// Mitsubishi GX Works2 project: 0926최신화dev   PLC: Q02U

PROGRAM INPUT
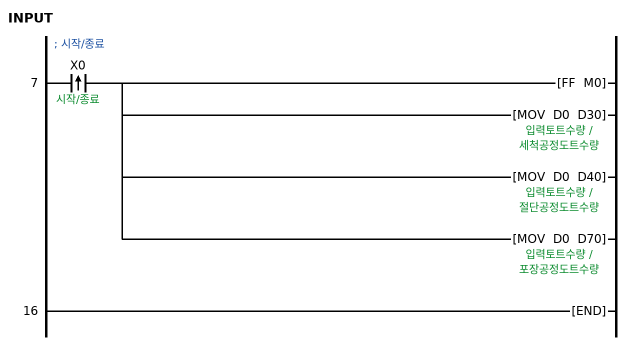
; 시작/종료
7     LDP     X0  ; 시작/종료
      FF      M0
      MOV     D0 D30  ; 입력토트수량 / 세척공정도트수량
      MOV     D0 D40  ; 절단공정도트수량
      MOV     D0 D70  ; 포장공정도트수량
16    END
END_PROGRAM

PROGRAM 세척공정
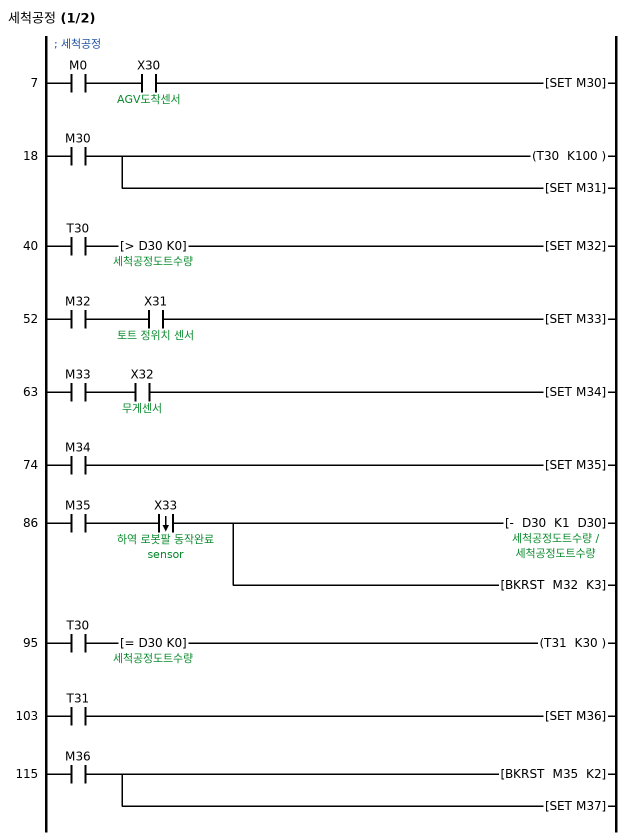
; 세척공정
7     LD      M0
      AND     X30  ; AGV도착센서
      SET     M30
        [note] 펌프모터 ON
18    LD      M30
      OUT     T30 K100
        [note] 펌핑모터 OFF
      SET     M31
        [note] SubCVY ON
40    LD      T30
      AND>    D30 K0  ; 세척공정도트수량
      SET     M32
        [note] 토트 발생
52    LD      M32
      AND     X31  ; 토트 정위치 센서
      SET     M33
        [note] MainCVY ON
63    LD      M33
      AND     X32  ; 무게센서
      SET     M34
        [note] MainCVY OFF
74    LD      M34
      SET     M35
        [note] 하역 로봇팔 ON
86    LD      M35
      ANDF    X33  ; 하역 로봇팔 동작완료 sensor
      -       D30 K1 D30
      BKRST   M32 K3
95    LD      T30
      AND=    D30 K0  ; 세척공정도트수량
      OUT     T31 K30
103   LD      T31
      SET     M36
        [note] 하역 로봇팔 OFF
115   LD      M36
      BKRST   M35 K2
      SET     M37
        [note] AGV 다음 공정 이동, SubCVY OFF
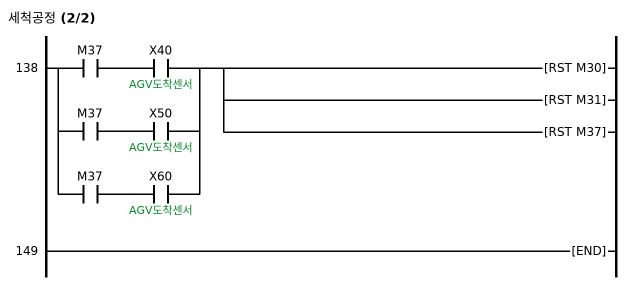
138   LD      M37
      AND     X40  ; AGV도착센서
      LD      M37
      AND     X50  ; AGV도착센서
      ORB
      LD      M37
      AND     X60  ; AGV도착센서
      ORB
      RST     M30
      RST     M31
      RST     M37
149   END
END_PROGRAM

PROGRAM 열풍건조
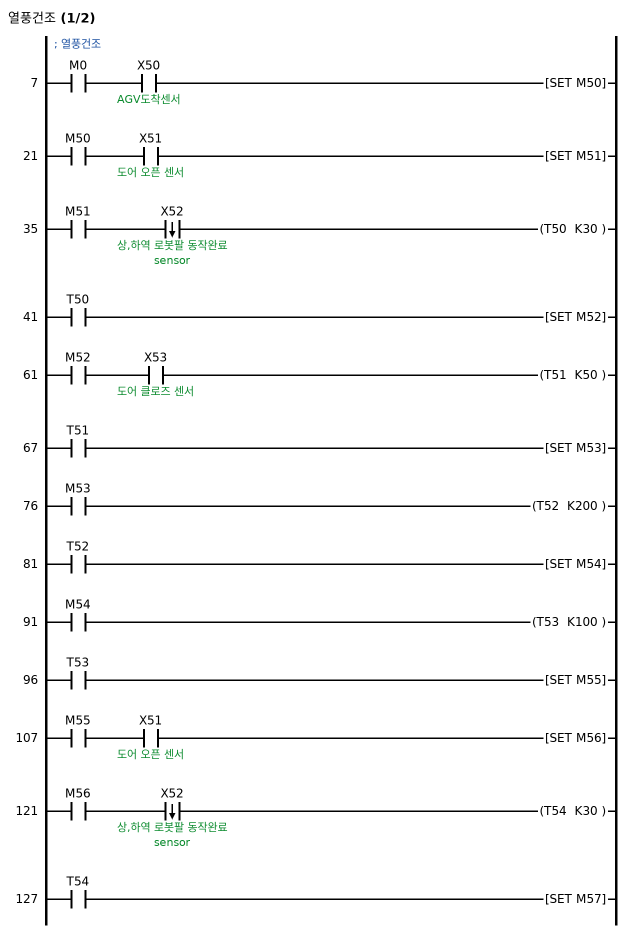
; 열풍건조
7     LD      M0
      AND     X50  ; AGV도착센서
      SET     M50
        [note] 도어 오픈모터(정)
21    LD      M50
      AND     X51  ; 도어 오픈 센서
      SET     M51
        [note] 상역 로봇 팔동작
35    LD      M51
      ANDF    X52  ; 상,하역 로봇팔 동작완료 sensor
      OUT     T50 K30
41    LD      T50
      SET     M52
        [note] 도어 클로즈모터(정), 로봇팔 OFF
61    LD      M52
      AND     X53  ; 도어 클로즈 센서
      OUT     T51 K50
67    LD      T51
      SET     M53
        [note] 건조기 ON
76    LD      M53
      OUT     T52 K200
81    LD      T52
      SET     M54
        [note] 건조기 OFF
91    LD      M54
      OUT     T53 K100
96    LD      T53
      SET     M55
        [note] 도어 오픈CYL
107   LD      M55
      AND     X51  ; 도어 오픈 센서
      SET     M56
        [note] 하역 로봇팔 동작
121   LD      M56
      ANDF    X52  ; 상,하역 로봇팔 동작완료 sensor
      OUT     T54 K30
127   LD      T54
      SET     M57
        [note] 도어 클로즈CYL, 로봇팔 OFF
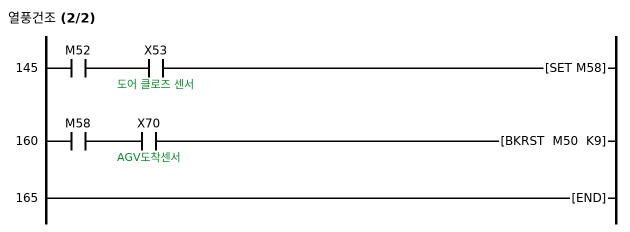
145   LD      M52
      AND     X53  ; 도어 클로즈 센서
      SET     M58
        [note] AGV 다음 공정 이동
160   LD      M58
      AND     X70  ; AGV도착센서
      BKRST   M50 K9
165   END
END_PROGRAM

PROGRAM OUTPUT
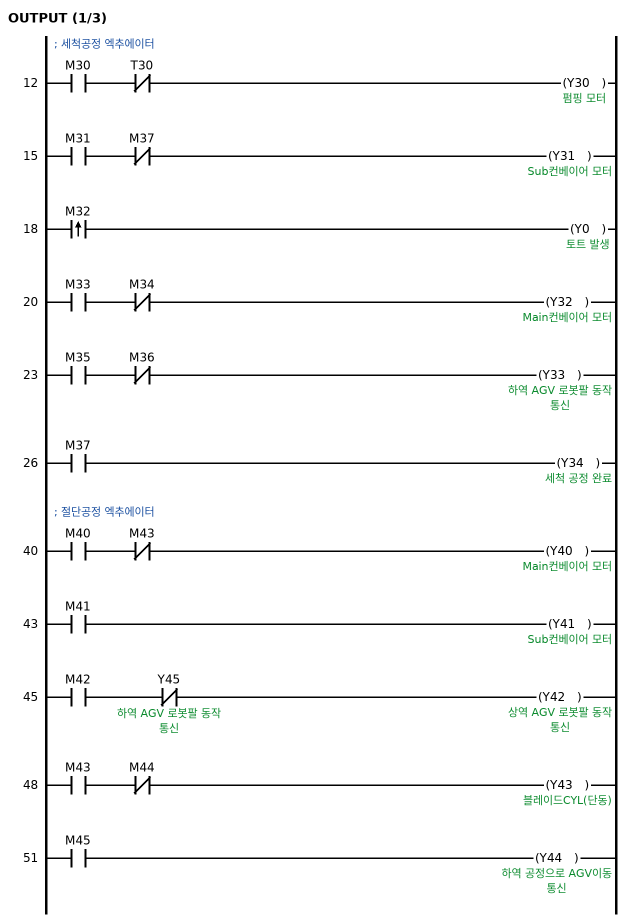
; 세척공정 엑추에이터
12    LD      M30
      ANI     T30
      OUT     Y30  ; 펌핑 모터
15    LD      M31
      ANI     M37
      OUT     Y31  ; Sub컨베이어 모터
18    LDP     M32
      OUT     Y0  ; 토트 발생
20    LD      M33
      ANI     M34
      OUT     Y32  ; Main컨베이어 모터
23    LD      M35
      ANI     M36
      OUT     Y33  ; 하역 AGV 로봇팔 동작 통신
26    LD      M37
      OUT     Y34  ; 세척 공정 완료
; 절단공정 엑추에이터
40    LD      M40
      ANI     M43
      OUT     Y40  ; Main컨베이어 모터
43    LD      M41
      OUT     Y41  ; Sub컨베이어 모터
45    LD      M42
      ANI     Y45  ; 하역 AGV 로봇팔 동작 통신
      OUT     Y42  ; 상역 AGV 로봇팔 동작 통신
48    LD      M43
      ANI     M44
      OUT     Y43  ; 블레이드CYL(단동)
51    LD      M45
      OUT     Y44  ; 하역 공정으로 AGV이동 통신
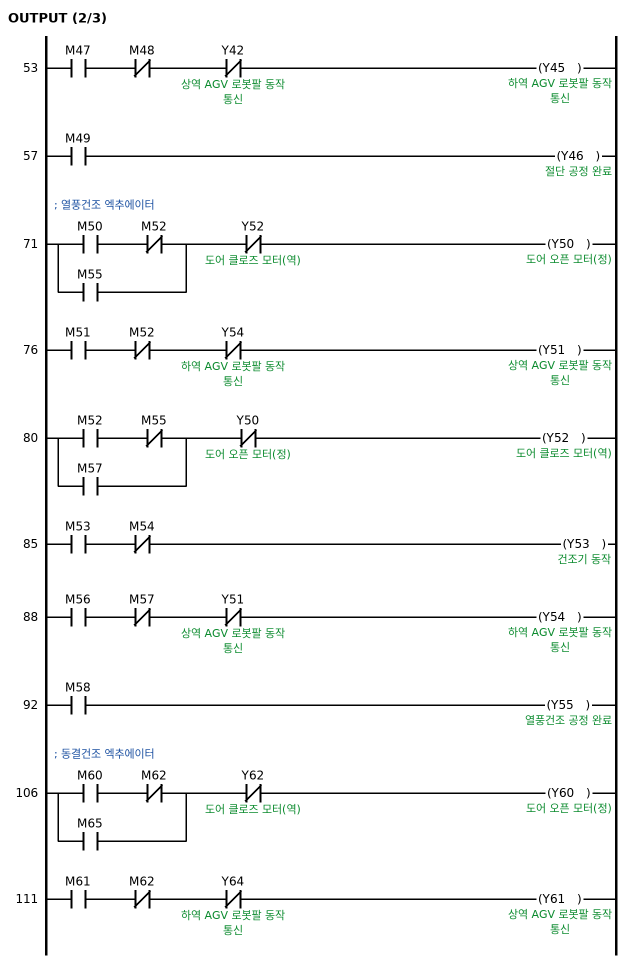
53    LD      M47
      ANI     M48
      ANI     Y42  ; 상역 AGV 로봇팔 동작 통신
      OUT     Y45  ; 하역 AGV 로봇팔 동작 통신
57    LD      M49
      OUT     Y46  ; 절단 공정 완료
; 열풍건조 엑추에이터
71    LD      M50
      ANI     M52
      OR      M55
      ANI     Y52  ; 도어 클로즈 모터(역)
      OUT     Y50  ; 도어 오픈 모터(정)
76    LD      M51
      ANI     M52
      ANI     Y54  ; 하역 AGV 로봇팔 동작 통신
      OUT     Y51  ; 상역 AGV 로봇팔 동작 통신
80    LD      M52
      ANI     M55
      OR      M57
      ANI     Y50  ; 도어 오픈 모터(정)
      OUT     Y52  ; 도어 클로즈 모터(역)
85    LD      M53
      ANI     M54
      OUT     Y53  ; 건조기 동작
88    LD      M56
      ANI     M57
      ANI     Y51  ; 상역 AGV 로봇팔 동작 통신
      OUT     Y54  ; 하역 AGV 로봇팔 동작 통신
92    LD      M58
      OUT     Y55  ; 열풍건조 공정 완료
; 동결건조 엑추에이터
106   LD      M60
      ANI     M62
      OR      M65
      ANI     Y62  ; 도어 클로즈 모터(역)
      OUT     Y60  ; 도어 오픈 모터(정)
111   LD      M61
      ANI     M62
      ANI     Y64  ; 하역 AGV 로봇팔 동작 통신
      OUT     Y61  ; 상역 AGV 로봇팔 동작 통신
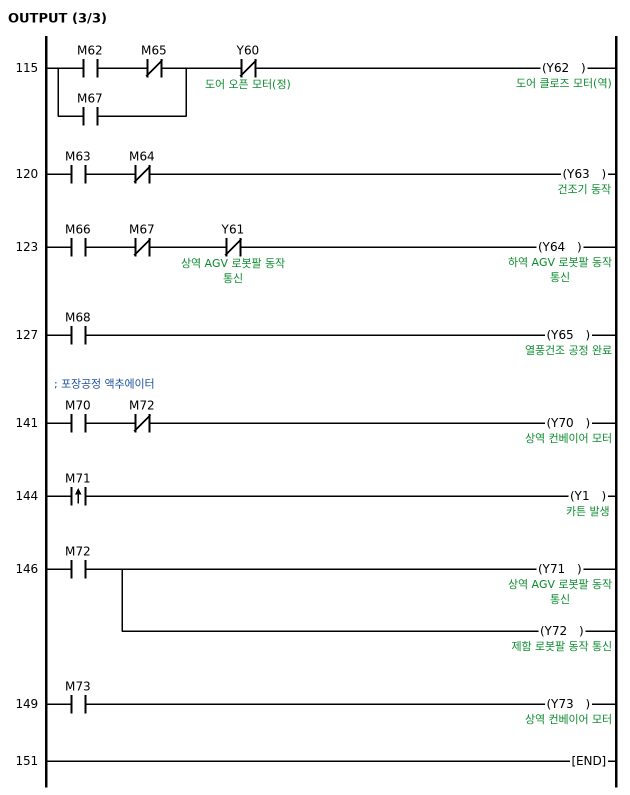
115   LD      M62
      ANI     M65
      OR      M67
      ANI     Y60  ; 도어 오픈 모터(정)
      OUT     Y62  ; 도어 클로즈 모터(역)
120   LD      M63
      ANI     M64
      OUT     Y63  ; 건조기 동작
123   LD      M66
      ANI     M67
      ANI     Y61  ; 상역 AGV 로봇팔 동작 통신
      OUT     Y64  ; 하역 AGV 로봇팔 동작 통신
127   LD      M68
      OUT     Y65  ; 열풍건조 공정 완료
; 포장공정 액추에이터
141   LD      M70
      ANI     M72
      OUT     Y70  ; 상역 컨베이어 모터
144   LDP     M71
      OUT     Y1  ; 카튼 발생
146   LD      M72
      OUT     Y71  ; 상역 AGV 로봇팔 동작 통신
      OUT     Y72  ; 제함 로봇팔 동작 통신
149   LD      M73
      OUT     Y73  ; 상역 컨베이어 모터
151   END
END_PROGRAM

PROGRAM 동결건조
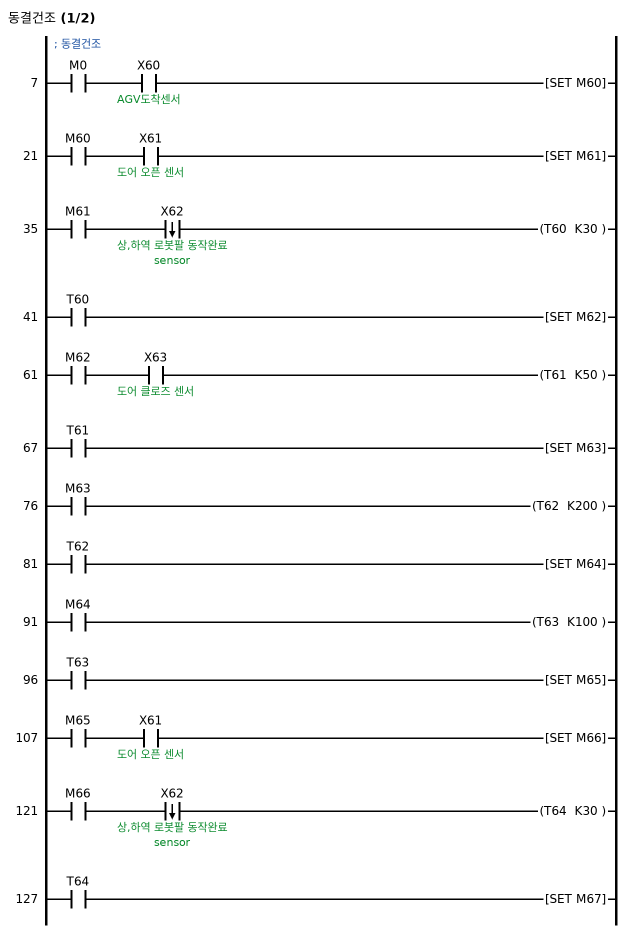
; 동결건조
7     LD      M0
      AND     X60  ; AGV도착센서
      SET     M60
        [note] 도어 오픈모터(정)
21    LD      M60
      AND     X61  ; 도어 오픈 센서
      SET     M61
        [note] 상역 로봇 팔동작
35    LD      M61
      ANDF    X62  ; 상,하역 로봇팔 동작완료 sensor
      OUT     T60 K30
41    LD      T60
      SET     M62
        [note] 도어 클로즈모터(정),로봇팔 OFF
61    LD      M62
      AND     X63  ; 도어 클로즈 센서
      OUT     T61 K50
67    LD      T61
      SET     M63
        [note] 건조기 ON
76    LD      M63
      OUT     T62 K200
81    LD      T62
      SET     M64
        [note] 건조기 OFF
91    LD      M64
      OUT     T63 K100
96    LD      T63
      SET     M65
        [note] 도어 오픈CYL
107   LD      M65
      AND     X61  ; 도어 오픈 센서
      SET     M66
        [note] 하역 로봇팔 동작
121   LD      M66
      ANDF    X62  ; 상,하역 로봇팔 동작완료 sensor
      OUT     T64 K30
127   LD      T64
      SET     M67
        [note] 도어 클로즈CYL, 로봇팔 OFF
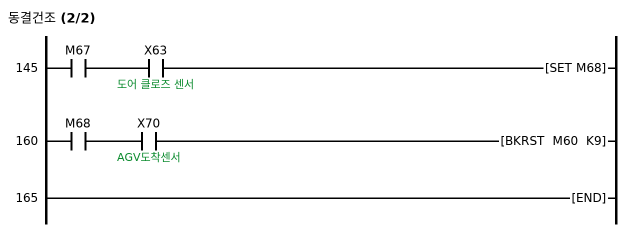
145   LD      M67
      AND     X63  ; 도어 클로즈 센서
      SET     M68
        [note] AGV 다음 공정 이동
160   LD      M68
      AND     X70  ; AGV도착센서
      BKRST   M60 K9
165   END
END_PROGRAM

PROGRAM 절단공정
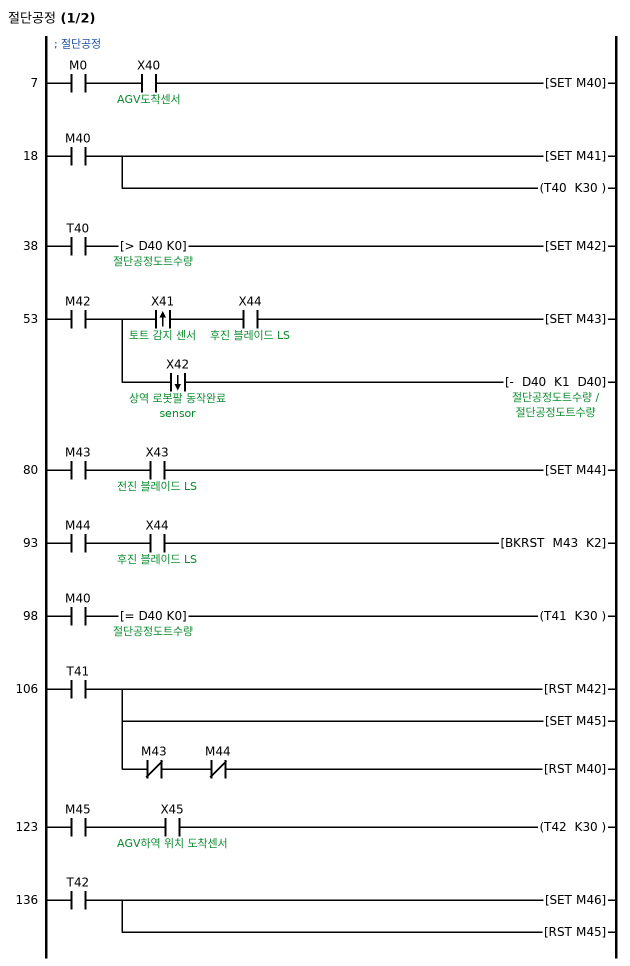
; 절단공정
7     LD      M0
      AND     X40  ; AGV도착센서
      SET     M40
        [note] MainCVY ON
18    LD      M40
      SET     M41
        [note] SubCVY ON
      OUT     T40 K30
        [note] 상역 여유
38    LD      T40
      AND>    D40 K0  ; 절단공정도트수량
      SET     M42
        [note] 상역 로봇팔 ON
53    LD      M42
      MPS
      ANDP    X41  ; 토트 감지 센서
      AND     X44  ; 후진 블레이드 LS
      SET     M43
        [note] MainCVY OFF, 블레이드CYL ON
      MPP
      ANDF    X42  ; 상역 로봇팔 동작완료 sensor
      -       D40 K1 D40
80    LD      M43
      AND     X43  ; 전진 블레이드 LS
      SET     M44
        [note] 블레이드CYL OFF
93    LD      M44
      AND     X44  ; 후진 블레이드 LS
      BKRST   M43 K2
98    LD      M40
      AND=    D40 K0  ; 절단공정도트수량
      OUT     T41 K30
106   LD      T41
      RST     M42
      SET     M45
        [note] AGV하역 위치 이동
      ANI     M43
      ANI     M44
      RST     M40
123   LD      M45
      AND     X45  ; AGV하역 위치 도착센서
      OUT     T42 K30
        [note] 하역 여유
136   LD      T42
      SET     M46
      RST     M45
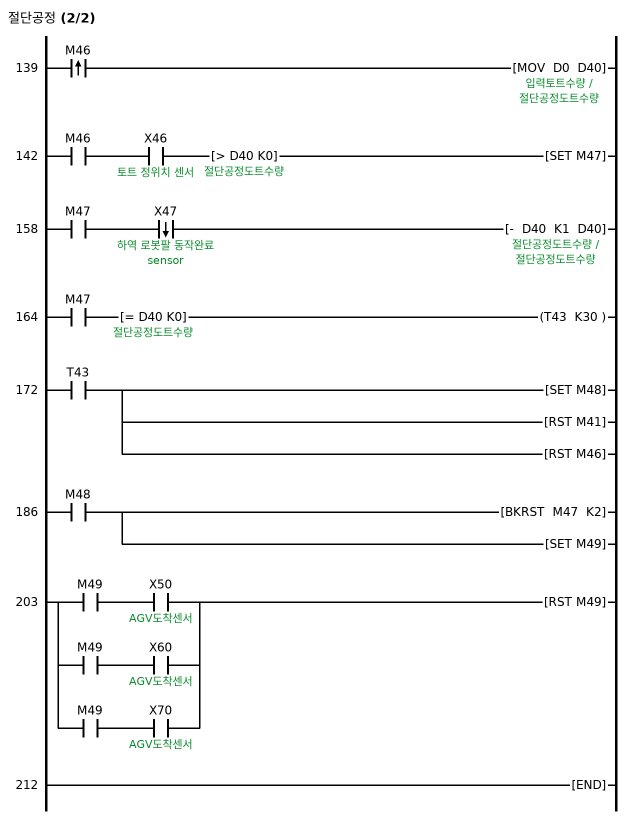
139   LDP     M46
      MOV     D0 D40  ; 입력토트수량
142   LD      M46
      AND     X46  ; 토트 정위치 센서
      AND>    D40 K0  ; 절단공정도트수량
      SET     M47
        [note] 하역 로봇팔 ON
158   LD      M47
      ANDF    X47  ; 하역 로봇팔 동작완료 sensor
      -       D40 K1 D40
164   LD      M47
      AND=    D40 K0  ; 절단공정도트수량
      OUT     T43 K30
172   LD      T43
      SET     M48
        [note] 하역 로봇팔 OFF
      RST     M41
      RST     M46
186   LD      M48
      BKRST   M47 K2
      SET     M49
        [note] AGV 다음 공정 이동
203   LD      M49
      AND     X50  ; AGV도착센서
      LD      M49
      AND     X60  ; AGV도착센서
      ORB
      LD      M49
      AND     X70  ; AGV도착센서
      ORB
      RST     M49
212   END
END_PROGRAM

PROGRAM 포장공정
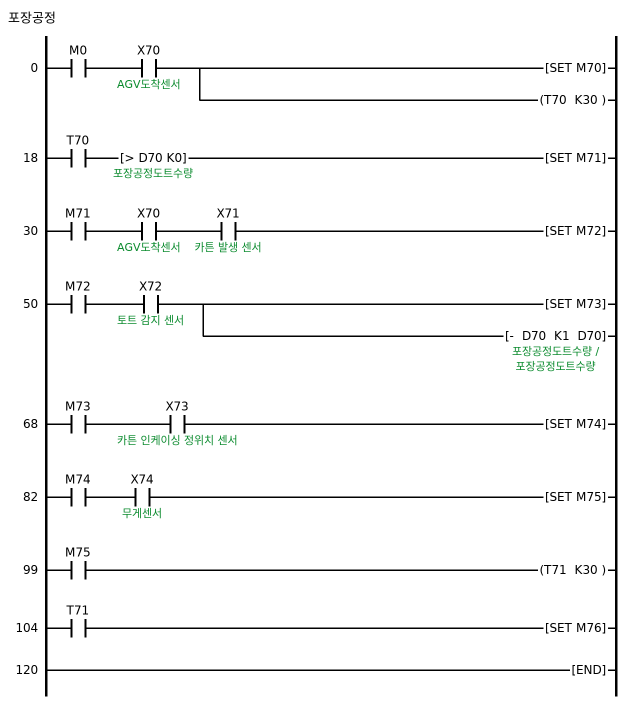
0     LD      M0
      AND     X70  ; AGV도착센서
      SET     M70
        [note] 상역 컨베이어 ON
      OUT     T70 K30
18    LD      T70
      AND>    D70 K0  ; 포장공정도트수량
      SET     M71
        [note] 카튼 발생
30    LD      M71
      AND     X70  ; AGV도착센서
      AND     X71  ; 카튼 발생 센서
      SET     M72
        [note] 상역 로봇팔, 제함 로봇팔 ON
50    LD      M72
      AND     X72  ; 토트 감지 센서
      SET     M73
        [note] 상역 컨베이어 OFF
      -       D70 K1 D70
68    LD      M73
      AND     X73  ; 카튼 인케이싱 정위치 센서
      SET     M74
        [note] 상역 컨벤이어 ON
82    LD      M74
      AND     X74  ; 무게센서
      SET     M75
        [note] 상부테이핑 컨베이어 ON
99    LD      M75
      OUT     T71 K30
104   LD      T71
      SET     M76
        [note] 상부테이핑 컨베이어 OFF
120   END
END_PROGRAM

// device comments not shown above
X75  ; 적재 스토퍼 센서
Y75  ; 상부 테이핑 컨베이어 모터1
Y76  ; 상부 테이핑 컨베이어 모터2
D50  ; 열풍건조공정도트수량
D60  ; 동결건조공정도트수량
